FUNCTION_BLOCK UNIT_OwnerLatch (* Local channel IDs of the occupation owner and its refresh query; types and forwards the received owner *)
  (* Standard: 61499-2 *)
  (* Version 0.1, 2026-09-28, Project contributors, AAU Smart Production Lab *)
  PACKAGE unitlib;
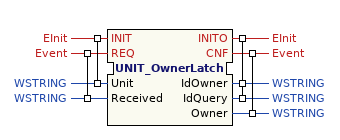
  EVENT_INPUT
    INIT : EInit WITH Unit;
    REQ WITH Received;
  END_EVENT
  EVENT_OUTPUT
    INITO : EInit WITH IdOwner, IdQuery;
    CNF WITH Owner;
  END_EVENT
  VAR_INPUT
    Unit : WSTRING;
    Received : WSTRING;
  END_VAR
  VAR_OUTPUT
    IdOwner : WSTRING;
    IdQuery : WSTRING;
    Owner : WSTRING;
  END_VAR
  EC_STATES
    INIT : INIT -> INITO;
    REQ : REQ -> CNF;
  END_STATES
  ALGORITHM INIT IN ST:
IdOwner := CONCAT(CONCAT("loc[", Unit), "/owner]");
IdQuery := CONCAT(CONCAT("loc[", Unit), "/owner/query]");
  END_ALGORITHM
  ALGORITHM REQ IN ST:
Owner := Received;
  END_ALGORITHM
END_FUNCTION_BLOCK
